(* IEC 61131-3 sources: RL_MAR/experiments/comparison/llm4plc/results/deepseek-ai-DeepSeek-V3.2_20260506_104945/20260506_120743, 4 files *)

(* ---- generated_code_iteration_0.st ---- *)
START_ST
FUNCTION_BLOCK PizzaMakingMachine
VAR_INPUT
    StartButton : BOOL;
    StopButton : BOOL;
    DoughReadySensor : BOOL;
    ToppingsReadySensor : BOOL;
    BakingDoneSensor : BOOL;
END_VAR

VAR_OUTPUT
    DoughRollerMotor : BOOL;
    ToppingDispenser : BOOL;
    ConveyorMotor : BOOL;
    OvenHeater : BOOL;
    OvenTemperature : INT;
END_VAR

VAR
    state : INT;
    prevState : INT;
    internalStopFlag : BOOL;
END_VAR

(* State Definitions *)
CONST
    STATE_IDLE := 0;
    STATE_ROLLING_DOUGH := 1;
    STATE_DISPENSING_TOPPINGS := 2;
    STATE_MOVING_TO_OVEN := 3;
    STATE_BAKING := 4;
    STATE_COOLING_OVEN := 5;
    STATE_EMERGENCY_STOP := 6;
END_CONST

(* Main Logic *)
IF StopButton THEN
    state := STATE_EMERGENCY_STOP;
    internalStopFlag := TRUE;
ELSIF internalStopFlag AND NOT StartButton THEN
    state := STATE_IDLE;
    internalStopFlag := FALSE;
ELSE
    CASE state OF
        STATE_IDLE:
            IF StartButton AND NOT StopButton THEN
                state := STATE_ROLLING_DOUGH;
            END_IF;

        STATE_ROLLING_DOUGH:
            IF DoughReadySensor THEN
                state := STATE_DISPENSING_TOPPINGS;
            END_IF;

        STATE_DISPENSING_TOPPINGS:
            IF ToppingsReadySensor THEN
                state := STATE_MOVING_TO_OVEN;
            END_IF;

        STATE_MOVING_TO_OVEN:
            IF NOT BakingDoneSensor THEN
                state := STATE_BAKING;
            END_IF;

        STATE_BAKING:
            IF BakingDoneSensor THEN
                state := STATE_COOLING_OVEN;
            END_IF;

        STATE_COOLING_OVEN:
            state := STATE_IDLE;

        STATE_EMERGENCY_STOP:
            (* Stay in emergency stop until conditions handled above *)
    END_CASE;
END_IF;

(* Store previous state for debugging/tracking *)
prevState := state;

(* Set outputs based on current state *)
CASE state OF
    STATE_IDLE:
        DoughRollerMotor := FALSE;
        ToppingDispenser := FALSE;
        ConveyorMotor := FALSE;
        OvenHeater := FALSE;
        OvenTemperature := 0;

    STATE_ROLLING_DOUGH:
        DoughRollerMotor := TRUE;
        ToppingDispenser := FALSE;
        ConveyorMotor := FALSE;
        OvenHeater := FALSE;
        OvenTemperature := 0;

    STATE_DISPENSING_TOPPINGS:
        DoughRollerMotor := FALSE;
        ToppingDispenser := TRUE;
        ConveyorMotor := FALSE;
        OvenHeater := FALSE;
        OvenTemperature := 0;

    STATE_MOVING_TO_OVEN:
        DoughRollerMotor := FALSE;
        ToppingDispenser := FALSE;
        ConveyorMotor := TRUE;
        OvenHeater := FALSE;
        OvenTemperature := 0;

    STATE_BAKING:
        DoughRollerMotor := FALSE;
        ToppingDispenser := FALSE;
        ConveyorMotor := FALSE;
        OvenHeater := TRUE;
        OvenTemperature := 220;

    STATE_COOLING_OVEN:
        DoughRollerMotor := FALSE;
        ToppingDispenser := FALSE;
        ConveyorMotor := FALSE;
        OvenHeater := FALSE;
        OvenTemperature := 0;

    STATE_EMERGENCY_STOP:
        DoughRollerMotor := FALSE;
        ToppingDispenser := FALSE;
        ConveyorMotor := FALSE;
        OvenHeater := FALSE;
        OvenTemperature := 0;
END_CASE;

END_FUNCTION_BLOCK
END_ST

(* ---- generated_code_iteration_1.st ---- *)
START_REASON
The feedback indicates a CODESYS compiler validation error: "应该用';' 替换'STATE_IDLE'". This is a Chinese error message meaning "should replace 'STATE_IDLE' with ';'". In CODESYS Structured Text, the CONST section requires each constant assignment to end with a semicolon (;), not a colon-equals (:=) followed by a semicolon. The current code uses "STATE_IDLE := 0;" which is incorrect for CODESYS. In CODESYS, constants are defined with "STATE_IDLE : INT := 0;" (with a colon, not colon-equals). However, the error message suggests replacing 'STATE_IDLE' with ';', which might be a misinterpretation—likely, the issue is the syntax of the constant definition. In CODESYS ST, the correct syntax for constants within a FUNCTION_BLOCK is to declare them in the VAR_CONSTANT section with proper type and assignment using ":=". The current code uses "CONST ... END_CONST" with ":=" which is not standard CODESYS. I need to change the constant definitions to use VAR_CONSTANT with proper syntax. Also, ensure all variable sections are closed with END_VAR, not END_VAR_INPUT or END_VAR_OUTPUT, which is already correct in the code. I'll adjust the constant definitions to comply with CODESYS standards.
END_REASON

START_ST
FUNCTION_BLOCK PizzaMakingMachine
VAR_INPUT
    StartButton : BOOL;
    StopButton : BOOL;
    DoughReadySensor : BOOL;
    ToppingsReadySensor : BOOL;
    BakingDoneSensor : BOOL;
END_VAR

VAR_OUTPUT
    DoughRollerMotor : BOOL;
    ToppingDispenser : BOOL;
    ConveyorMotor : BOOL;
    OvenHeater : BOOL;
    OvenTemperature : INT;
END_VAR

VAR
    state : INT;
    prevState : INT;
    internalStopFlag : BOOL;
END_VAR

VAR_CONSTANT
    STATE_IDLE : INT := 0;
    STATE_ROLLING_DOUGH : INT := 1;
    STATE_DISPENSING_TOPPINGS : INT := 2;
    STATE_MOVING_TO_OVEN : INT := 3;
    STATE_BAKING : INT := 4;
    STATE_COOLING_OVEN : INT := 5;
    STATE_EMERGENCY_STOP : INT := 6;
END_VAR

(* Main Logic *)
IF StopButton THEN
    state := STATE_EMERGENCY_STOP;
    internalStopFlag := TRUE;
ELSIF internalStopFlag AND NOT StartButton THEN
    state := STATE_IDLE;
    internalStopFlag := FALSE;
ELSE
    CASE state OF
        STATE_IDLE:
            IF StartButton AND NOT StopButton THEN
                state := STATE_ROLLING_DOUGH;
            END_IF;

        STATE_ROLLING_DOUGH:
            IF DoughReadySensor THEN
                state := STATE_DISPENSING_TOPPINGS;
            END_IF;

        STATE_DISPENSING_TOPPINGS:
            IF ToppingsReadySensor THEN
                state := STATE_MOVING_TO_OVEN;
            END_IF;

        STATE_MOVING_TO_OVEN:
            IF NOT BakingDoneSensor THEN
                state := STATE_BAKING;
            END_IF;

        STATE_BAKING:
            IF BakingDoneSensor THEN
                state := STATE_COOLING_OVEN;
            END_IF;

        STATE_COOLING_OVEN:
            state := STATE_IDLE;

        STATE_EMERGENCY_STOP:
            (* Stay in emergency stop until conditions handled above *)
    END_CASE;
END_IF;

(* Store previous state for debugging/tracking *)
prevState := state;

(* Set outputs based on current state *)
CASE state OF
    STATE_IDLE:
        DoughRollerMotor := FALSE;
        ToppingDispenser := FALSE;
        ConveyorMotor := FALSE;
        OvenHeater := FALSE;
        OvenTemperature := 0;

    STATE_ROLLING_DOUGH:
        DoughRollerMotor := TRUE;
        ToppingDispenser := FALSE;
        ConveyorMotor := FALSE;
        OvenHeater := FALSE;
        OvenTemperature := 0;

    STATE_DISPENSING_TOPPINGS:
        DoughRollerMotor := FALSE;
        ToppingDispenser := TRUE;
        ConveyorMotor := FALSE;
        OvenHeater := FALSE;
        OvenTemperature := 0;

    STATE_MOVING_TO_OVEN:
        DoughRollerMotor := FALSE;
        ToppingDispenser := FALSE;
        ConveyorMotor := TRUE;
        OvenHeater := FALSE;
        OvenTemperature := 0;

    STATE_BAKING:
        DoughRollerMotor := FALSE;
        ToppingDispenser := FALSE;
        ConveyorMotor := FALSE;
        OvenHeater := TRUE;
        OvenTemperature := 220;

    STATE_COOLING_OVEN:
        DoughRollerMotor := FALSE;
        ToppingDispenser := FALSE;
        ConveyorMotor := FALSE;
        OvenHeater := FALSE;
        OvenTemperature := 0;

    STATE_EMERGENCY_STOP:
        DoughRollerMotor := FALSE;
        ToppingDispenser := FALSE;
        ConveyorMotor := FALSE;
        OvenHeater := FALSE;
        OvenTemperature := 0;
END_CASE;

END_FUNCTION_BLOCK
END_ST

(* ---- generated_code_iteration_2.st ---- *)
START_REASON
The feedback indicates an encoding issue: "gbk codec can't decode byte 0xaf in position 79: illegal multibyte sequence." This error occurs because the code contains non-ASCII characters that cannot be decoded with the GBK encoding used by the CODESYS compiler. In the previous code, the comment "(* Main Logic *)" and other comments might contain special characters or the issue could be with the Chinese error message in the feedback itself. However, since the feedback is about the code validation, I need to ensure the ST code uses only ASCII characters and proper syntax. The error mentions position 79, which likely points to a specific character in the code. I'll review the code for any non-ASCII characters, such as in comments or strings, and replace them with ASCII equivalents. Also, I'll ensure all syntax is correct for CODESYS, including constant definitions and variable sections. The previous fix already adjusted constants to VAR_CONSTANT, but I'll double-check for any hidden non-ASCII characters (e.g., in comments or variable names). I'll rewrite the code with ASCII-only comments and ensure no special characters are present.
END_REASON

START_ST
FUNCTION_BLOCK PizzaMakingMachine
VAR_INPUT
    StartButton : BOOL;
    StopButton : BOOL;
    DoughReadySensor : BOOL;
    ToppingsReadySensor : BOOL;
    BakingDoneSensor : BOOL;
END_VAR

VAR_OUTPUT
    DoughRollerMotor : BOOL;
    ToppingDispenser : BOOL;
    ConveyorMotor : BOOL;
    OvenHeater : BOOL;
    OvenTemperature : INT;
END_VAR

VAR
    state : INT;
    prevState : INT;
    internalStopFlag : BOOL;
END_VAR

VAR_CONSTANT
    STATE_IDLE : INT := 0;
    STATE_ROLLING_DOUGH : INT := 1;
    STATE_DISPENSING_TOPPINGS : INT := 2;
    STATE_MOVING_TO_OVEN : INT := 3;
    STATE_BAKING : INT := 4;
    STATE_COOLING_OVEN : INT := 5;
    STATE_EMERGENCY_STOP : INT := 6;
END_VAR

(* Main Logic *)
IF StopButton THEN
    state := STATE_EMERGENCY_STOP;
    internalStopFlag := TRUE;
ELSIF internalStopFlag AND NOT StartButton THEN
    state := STATE_IDLE;
    internalStopFlag := FALSE;
ELSE
    CASE state OF
        STATE_IDLE:
            IF StartButton AND NOT StopButton THEN
                state := STATE_ROLLING_DOUGH;
            END_IF;

        STATE_ROLLING_DOUGH:
            IF DoughReadySensor THEN
                state := STATE_DISPENSING_TOPPINGS;
            END_IF;

        STATE_DISPENSING_TOPPINGS:
            IF ToppingsReadySensor THEN
                state := STATE_MOVING_TO_OVEN;
            END_IF;

        STATE_MOVING_TO_OVEN:
            IF NOT BakingDoneSensor THEN
                state := STATE_BAKING;
            END_IF;

        STATE_BAKING:
            IF BakingDoneSensor THEN
                state := STATE_COOLING_OVEN;
            END_IF;

        STATE_COOLING_OVEN:
            state := STATE_IDLE;

        STATE_EMERGENCY_STOP:
            (* Stay in emergency stop until conditions handled above *)
    END_CASE;
END_IF;

(* Store previous state for debugging *)
prevState := state;

(* Set outputs based on current state *)
CASE state OF
    STATE_IDLE:
        DoughRollerMotor := FALSE;
        ToppingDispenser := FALSE;
        ConveyorMotor := FALSE;
        OvenHeater := FALSE;
        OvenTemperature := 0;

    STATE_ROLLING_DOUGH:
        DoughRollerMotor := TRUE;
        ToppingDispenser := FALSE;
        ConveyorMotor := FALSE;
        OvenHeater := FALSE;
        OvenTemperature := 0;

    STATE_DISPENSING_TOPPINGS:
        DoughRollerMotor := FALSE;
        ToppingDispenser := TRUE;
        ConveyorMotor := FALSE;
        OvenHeater := FALSE;
        OvenTemperature := 0;

    STATE_MOVING_TO_OVEN:
        DoughRollerMotor := FALSE;
        ToppingDispenser := FALSE;
        ConveyorMotor := TRUE;
        OvenHeater := FALSE;
        OvenTemperature := 0;

    STATE_BAKING:
        DoughRollerMotor := FALSE;
        ToppingDispenser := FALSE;
        ConveyorMotor := FALSE;
        OvenHeater := TRUE;
        OvenTemperature := 220;

    STATE_COOLING_OVEN:
        DoughRollerMotor := FALSE;
        ToppingDispenser := FALSE;
        ConveyorMotor := FALSE;
        OvenHeater := FALSE;
        OvenTemperature := 0;

    STATE_EMERGENCY_STOP:
        DoughRollerMotor := FALSE;
        ToppingDispenser := FALSE;
        ConveyorMotor := FALSE;
        OvenHeater := FALSE;
        OvenTemperature := 0;
END_CASE;

END_FUNCTION_BLOCK
END_ST

(* ---- generated_code_iteration_3.st ---- *)
START_REASON
The feedback indicates that the CODESYS compiler validation failed because VAR_CONSTANT is not allowed in the current context. In CODESYS Structured Text, constants should be defined using the CONSTANT keyword directly, not within a VAR_CONSTANT section. The error message "应该采用VAR, VAR_INPUT, VAR_OUTPUT 或 VAR_IN_OUT 取代VAR_CONSTANT" suggests replacing VAR_CONSTANT with one of the standard variable sections. To fix this, I need to change the constant definitions to use the correct syntax: either define them as global constants outside the FUNCTION_BLOCK or use proper constant declarations within the block. Since the constants are specific to this function block, I'll define them as local constants using the correct CODESYS syntax. In CODESYS, constants in a function block are typically declared with "CONSTANT" without the VAR prefix. I'll adjust the code accordingly to comply with CODESYS standards.
END_REASON

START_ST
FUNCTION_BLOCK PizzaMakingMachine
VAR_INPUT
    StartButton : BOOL;
    StopButton : BOOL;
    DoughReadySensor : BOOL;
    ToppingsReadySensor : BOOL;
    BakingDoneSensor : BOOL;
END_VAR

VAR_OUTPUT
    DoughRollerMotor : BOOL;
    ToppingDispenser : BOOL;
    ConveyorMotor : BOOL;
    OvenHeater : BOOL;
    OvenTemperature : INT;
END_VAR

VAR
    state : INT;
    prevState : INT;
    internalStopFlag : BOOL;
END_VAR

CONSTANT
    STATE_IDLE : INT := 0;
    STATE_ROLLING_DOUGH : INT := 1;
    STATE_DISPENSING_TOPPINGS : INT := 2;
    STATE_MOVING_TO_OVEN : INT := 3;
    STATE_BAKING : INT := 4;
    STATE_COOLING_OVEN : INT := 5;
    STATE_EMERGENCY_STOP : INT := 6;
END_CONSTANT

(* Main Logic *)
IF StopButton THEN
    state := STATE_EMERGENCY_STOP;
    internalStopFlag := TRUE;
ELSIF internalStopFlag AND NOT StartButton THEN
    state := STATE_IDLE;
    internalStopFlag := FALSE;
ELSE
    CASE state OF
        STATE_IDLE:
            IF StartButton AND NOT StopButton THEN
                state := STATE_ROLLING_DOUGH;
            END_IF;

        STATE_ROLLING_DOUGH:
            IF DoughReadySensor THEN
                state := STATE_DISPENSING_TOPPINGS;
            END_IF;

        STATE_DISPENSING_TOPPINGS:
            IF ToppingsReadySensor THEN
                state := STATE_MOVING_TO_OVEN;
            END_IF;

        STATE_MOVING_TO_OVEN:
            IF NOT BakingDoneSensor THEN
                state := STATE_BAKING;
            END_IF;

        STATE_BAKING:
            IF BakingDoneSensor THEN
                state := STATE_COOLING_OVEN;
            END_IF;

        STATE_COOLING_OVEN:
            state := STATE_IDLE;

        STATE_EMERGENCY_STOP:
            (* Stay in emergency stop until conditions handled above *)
    END_CASE;
END_IF;

(* Store previous state for debugging *)
prevState := state;

(* Set outputs based on current state *)
CASE state OF
    STATE_IDLE:
        DoughRollerMotor := FALSE;
        ToppingDispenser := FALSE;
        ConveyorMotor := FALSE;
        OvenHeater := FALSE;
        OvenTemperature := 0;

    STATE_ROLLING_DOUGH:
        DoughRollerMotor := TRUE;
        ToppingDispenser := FALSE;
        ConveyorMotor := FALSE;
        OvenHeater := FALSE;
        OvenTemperature := 0;

    STATE_DISPENSING_TOPPINGS:
        DoughRollerMotor := FALSE;
        ToppingDispenser := TRUE;
        ConveyorMotor := FALSE;
        OvenHeater := FALSE;
        OvenTemperature := 0;

    STATE_MOVING_TO_OVEN:
        DoughRollerMotor := FALSE;
        ToppingDispenser := FALSE;
        ConveyorMotor := TRUE;
        OvenHeater := FALSE;
        OvenTemperature := 0;

    STATE_BAKING:
        DoughRollerMotor := FALSE;
        ToppingDispenser := FALSE;
        ConveyorMotor := FALSE;
        OvenHeater := TRUE;
        OvenTemperature := 220;

    STATE_COOLING_OVEN:
        DoughRollerMotor := FALSE;
        ToppingDispenser := FALSE;
        ConveyorMotor := FALSE;
        OvenHeater := FALSE;
        OvenTemperature := 0;

    STATE_EMERGENCY_STOP:
        DoughRollerMotor := FALSE;
        ToppingDispenser := FALSE;
        ConveyorMotor := FALSE;
        OvenHeater := FALSE;
        OvenTemperature := 0;
END_CASE;

END_FUNCTION_BLOCK
END_ST
